PROGRAM MAIN
VAR
END_VAR

IO._CX2040.Run();

END_PROGRAM

(* stored: Version 1.1.0.1, ProductVersion 3.1.4024.9
   POU MAIN: Id {9bf4adaf-0f2d-0ac2-2cb1-948afa0b8cdf}, SpecialFunc None *)
